// TIA Portal V16 export
// export: Created 2022-07-21T09:35:28.3226111Z, ExportSetting WithDefaults, DisplayName Totally Integrated Automation Portal, DisplayVersion V16 Update 4, DisplayName TIA Portal Version Control Interface, DisplayVersion V16 Update 2, DisplayName TIA Portal Openness, DisplayVersion V16 Update 4, DisplayName SINAMICS Startdrive Advanced, DisplayVersion V16 Update 5, DisplayName SINAMICS Startdrive G130, G150, S120, S150, SINAMICS MV, S210, DisplayVersion V16 Update 5, DisplayName SINAMICS Startdrive G110M, G120, G120C, G120D, G120P, G115D, DisplayVersion V16 Update 5, DisplayName STEP 7 Professional, DisplayVersion V16 Update 4, DisplayName STEP 7 Safety, DisplayVersion V16, DisplayName WinCC Advanced, DisplayVersion V16 Update 4
FUNCTION_BLOCK "fbDriveSiemens"   // FB706, LAD
TITLE = Drive Siemens
{ S7_Optimized_Access := 'TRUE' }
VERSION : 0.1
// stored: AutoNumber false, IsIECCheckEnabled false, IsRetainMemResEnabled false, MemoryReserve 100, SetENOAutomatically false, UDAEnableTagReadback false
   VAR_INPUT
      executeAbslute : Bool;   // Ruch do zadanej pozycji / Move to preset position
      executeRelative : Bool;   // Przesunięcie o zadaną pozycję / Move by preset position
      stop : Bool;   // stop
      extAlm : Bool;   // zewnętrzny alarm / external alarm
      velocityAuto : LReal;   // [mm/s]
      velocityMan : LReal;   // [mm/s]
      acceleration : LReal;   // [mm/s²]
      decceleration : LReal;   // [mm/s²]
      group : "typeGroup";
      axis : TO_PositioningAxis;
   END_VAR
   VAR_IN_OUT
      drive : "typeDrive";
      axisBasicsDataBlock : "LAxisBasics_typeAxisBasicsData";
      axisConfiguration : "LAxisCtrl_typeAxisConfig";
   END_VAR
   VAR
      delayPTAlm0 : Time := T#1s;   // Czas opóźnienia dla alarmu 0 / delay alarm 0
      delayPTAlm1 : Time := T#1s;   // Czas opóźnienia dla alarmu 1 / delay alarm 1
      delayPTAlm2 : Time := T#1s;   // Czas opóźnienia dla alarmu 2 / delay alarm 2
      delayPTAlm3 : Time := T#1s;   // Czas opóźnienia dla alarmu 3 / delay alarm 3
      delayPTAlm4 : Time := T#1s;   // Czas opóźnienia dla alarmu 4 / delay alarm 4
      delayPTAlm5 : Time := T#1s;   // Czas opóźnienia dla alarmu 5 / delay alarm 5
      delayPTAlm6 : Time := T#1s;   // Czas opóźnienia dla alarmu 6 / delay alarm 6
      delayPTAlm7 : Time := T#1s;   // Czas opóźnienia dla alarmu 7 / delay alarm 7
      instTmrDlyAlm0 { S7_SetPoint := 'True'} : TON_TIME;   // Opóźnienie dla alarmu 0 / delay alarm 0
      instTmrDlyAlm1 { S7_SetPoint := 'True'} : TON_TIME;   // Opóźnienie dla alarmu 1 / delay alarm 1
      instTmrDlyAlm2 { S7_SetPoint := 'True'} : TON_TIME;   // Opóźnienie dla alarmu 2 / delay alarm 2
      instTmrDlyAlm3 { S7_SetPoint := 'True'} : TON_TIME;   // Opóźnienie dla alarmu 3 / delay alarm 3
      instTmrDlyAlm4 { S7_SetPoint := 'True'} : TON_TIME;   // Opóźnienie dla alarmu 4 / delay alarm 4
      instTmrDlyAlm5 { S7_SetPoint := 'True'} : TON_TIME;   // Opóźnienie dla alarmu 5 / delay alarm 5
      instTmrDlyAlm6 { S7_SetPoint := 'True'} : TON_TIME;   // Opóźnienie dla alarmu 6 / delay alarm 6
      instTmrDlyAlm7 { S7_SetPoint := 'True'} : TON_TIME;   // Opóźnienie dla alarmu 7 / delay alarm 7
      instLAxisCtrl_PosAxis { S7_SetPoint := 'True'} : "LAxisCtrl_PosAxis";
      instSetpointVelocity { S7_SetPoint := 'True'} : "fbSPEntryLReal";
      instSetpointPosition { S7_SetPoint := 'True'} : "fbSPEntryLReal";
      statOldAuto { S7_SetPoint := 'True'} : Bool;
      statOldMan : Bool;
      homePulse { S7_SetPoint := 'True'} : TP_TIME;
      instCompPosHome { S7_SetPoint := 'True'} : "fbCompareLReal";   // Porównanie pozycji domowej oś Z / Compare home position Z axis
   END_VAR
   VAR_TEMP
      bAlm0 : Bool;   // tymczasowy bit dla alarmu 0 / temporary alarm bit 0
      bAlm1 : Bool;   // tymczasowy bit dla alarmu 1 / temporary alarm bit 1
      bAlm2 : Bool;   // tymczasowy bit dla alarmu 2 / temporary alarm bit 2
      bAlm3 : Bool;   // tymczasowy bit dla alarmu 3 / temporary alarm bit 3
      bAlm4 : Bool;   // tymczasowy bit dla alarmu 4 / temporary alarm bit 4
      bAlm5 : Bool;   // tymczasowy bit dla alarmu 5 / temporary alarm bit 5
      bAlm6 : Bool;   // tymczasowy bit dla alarmu 6 / temporary alarm bit 6
      bAlm7 : Bool;   // tymczasowy bit dla alarmu 7 / temporary alarm bit 7
      seqStart : Bool;
      "robot in cv zone" : Bool;
   END_VAR
   VAR CONSTANT
      MAX_VEL_AUTO : LReal := 2000.0;   // prędkość w trybie automatycznym / speed in automatic mode
      MAX_VEL_MAN : LReal := 2000.0;
      MIN_VEL : LReal := 0.1;
      MIN_DIST : LReal := -1000.0;
      MAX_DIST : LReal := 5000.0;
   END_VAR
BEGIN

REGION Network 1: Alarm: axis error / Alarm: błąd osi
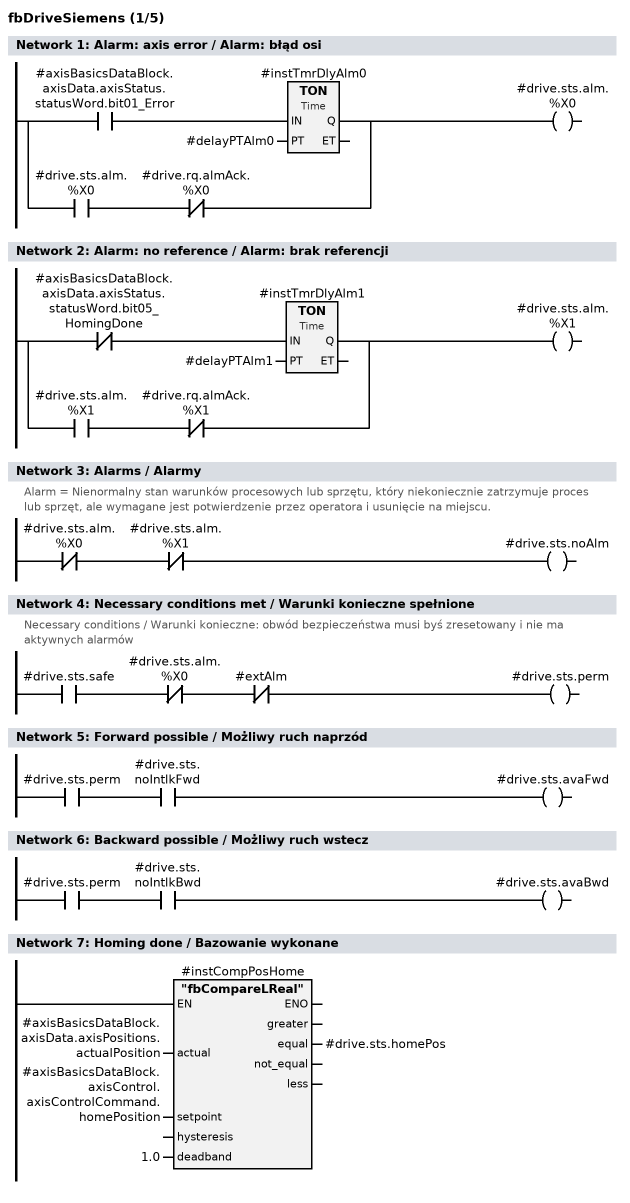
   RUNG wire#powerrail
      Contact( #axisBasicsDataBlock.axisData.axisStatus.statusWord.bit01_Error )
      { S7_Templates := "time_type := Time" } #instTmrDlyAlm0.TON(pt := #delayPTAlm0, et =>)
      wire#w1
      Coil( #drive.sts.alm.%X0 )
   END_RUNG
   RUNG wire#powerrail
      Contact( #drive.sts.alm.%X0 )
      I_Contact( #drive.rq.almAck.%X0 )
   END_RUNG wire#w1
   // the same network as SCL:
   #instTmrDlyAlm0(IN := #axisBasicsDataBlock.axisData.axisStatus.statusWord.bit01_Error, PT := #delayPTAlm0);   // TON
   #drive.sts.alm.%X0 := #instTmrDlyAlm0.Q OR (#drive.sts.alm.%X0 AND NOT #drive.rq.almAck.%X0);
END_REGION

REGION Network 2: Alarm: no reference / Alarm: brak referencji
   RUNG wire#powerrail
      I_Contact( #axisBasicsDataBlock.axisData.axisStatus.statusWord.bit05_HomingDone )
      { S7_Templates := "time_type := Time" } #instTmrDlyAlm1.TON(pt := #delayPTAlm1, et =>)
      wire#w1
      Coil( #drive.sts.alm.%X1 )
   END_RUNG
   RUNG wire#powerrail
      Contact( #drive.sts.alm.%X1 )
      I_Contact( #drive.rq.almAck.%X1 )
   END_RUNG wire#w1
   // the same network as SCL:
   #instTmrDlyAlm1(IN := NOT #axisBasicsDataBlock.axisData.axisStatus.statusWord.bit05_HomingDone,   // TON
                   PT := #delayPTAlm1);
   #drive.sts.alm.%X1 := #instTmrDlyAlm1.Q OR (#drive.sts.alm.%X1 AND NOT #drive.rq.almAck.%X1);
END_REGION

REGION Network 3: Alarms / Alarmy
   // Alarm = Nienormalny stan warunków procesowych lub sprzętu, który niekoniecznie zatrzymuje proces lub sprzęt, ale wymagane jest potwierdzenie przez operatora i usunięcie na miejscu.
   RUNG wire#powerrail
      I_Contact( #drive.sts.alm.%X0 )
      I_Contact( #drive.sts.alm.%X1 )
      Coil( #drive.sts.noAlm )
   END_RUNG
   // the same network as SCL:
   #drive.sts.noAlm := NOT #drive.sts.alm.%X0 AND NOT #drive.sts.alm.%X1;
END_REGION

REGION Network 4: Necessary conditions met / Warunki konieczne spełnione
   // Necessary conditions / Warunki konieczne: obwód bezpieczeństwa musi byś zresetowany i nie ma aktywnych alarmów
   RUNG wire#powerrail
      Contact( #drive.sts.safe )
      I_Contact( #drive.sts.alm.%X0 )
      I_Contact( #extAlm )
      Coil( #drive.sts.perm )
   END_RUNG
   // the same network as SCL:
   #drive.sts.perm := #drive.sts.safe AND NOT #drive.sts.alm.%X0 AND NOT #extAlm;
END_REGION

REGION Network 5: Forward possible / Możliwy ruch naprzód
   RUNG wire#powerrail
      Contact( #drive.sts.perm )
      Contact( #drive.sts.noIntlkFwd )
      Coil( #drive.sts.avaFwd )
   END_RUNG
   // the same network as SCL:
   #drive.sts.avaFwd := #drive.sts.perm AND #drive.sts.noIntlkFwd;
END_REGION

REGION Network 6: Backward possible / Możliwy ruch wstecz
   RUNG wire#powerrail
      Contact( #drive.sts.perm )
      Contact( #drive.sts.noIntlkBwd )
      Coil( #drive.sts.avaBwd )
   END_RUNG
   // the same network as SCL:
   #drive.sts.avaBwd := #drive.sts.perm AND #drive.sts.noIntlkBwd;
END_REGION

REGION Network 7: Homing done / Bazowanie wykonane
   RUNG wire#powerrail
      #instCompPosHome(actual := #axisBasicsDataBlock.axisData.axisPositions.actualPosition, setpoint := #axisBasicsDataBlock.axisControl.axisControlCommand.homePosition, hysteresis :=, deadband := 1.0, greater =>, equal => #drive.sts.homePos, not_equal =>, less =>)
   END_RUNG
   // the same network as SCL:
   #instCompPosHome(actual := #axisBasicsDataBlock.axisData.axisPositions.actualPosition,   // "fbCompareLReal"
                    setpoint := #axisBasicsDataBlock.axisControl.axisControlCommand.homePosition,
                    deadband := 1.0,
                    equal => #drive.sts.homePos);
END_REGION

REGION Network 8: Enable / Zezwolenie
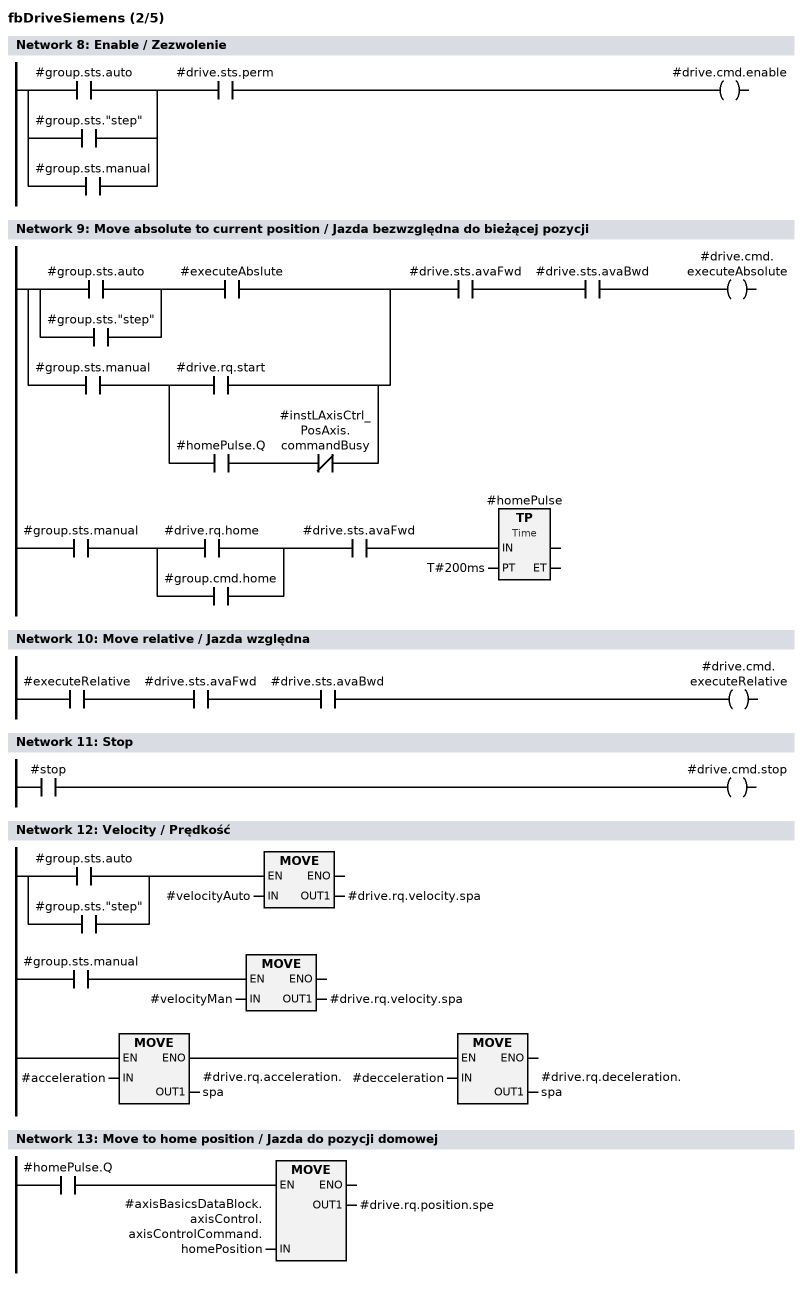
   RUNG wire#powerrail
      Contact( #group.sts.auto )
      wire#w1
      Contact( #drive.sts.perm )
      Coil( #drive.cmd.enable )
   END_RUNG
   RUNG wire#powerrail
      Contact( #group.sts."step" )
   END_RUNG wire#w1
   RUNG wire#powerrail
      Contact( #group.sts.manual )
   END_RUNG wire#w1
   // the same network as SCL:
   #drive.cmd.enable := (#group.sts.auto OR #group.sts."step" OR #group.sts.manual) AND #drive.sts.perm;
END_REGION

REGION Network 9: Move absolute to current position / Jazda bezwzględna do bieżącej pozycji
   RUNG wire#powerrail
      Contact( #group.sts.auto )
      wire#w1
      Contact( #executeAbslute )
      wire#w2
      Contact( #drive.sts.avaFwd )
      Contact( #drive.sts.avaBwd )
      Coil( #drive.cmd.executeAbsolute )
   END_RUNG
   RUNG wire#powerrail
      Contact( #group.sts."step" )
   END_RUNG wire#w1
   RUNG wire#powerrail
      Contact( #group.sts.manual )
      wire#w3
      Contact( #drive.rq.start )
   END_RUNG wire#w2
   RUNG wire#w3
      Contact( #homePulse.Q )
      I_Contact( #instLAxisCtrl_PosAxis.commandBusy )
   END_RUNG wire#w2
   RUNG wire#powerrail
      Contact( #group.sts.manual )
      wire#w4
      Contact( #drive.rq.home )
      wire#w5
      Contact( #drive.sts.avaFwd )
      { S7_Templates := "time_type := Time" } #homePulse.TP(pt := T#200ms, et =>)
   END_RUNG
   RUNG wire#w4
      Contact( #group.cmd.home )
   END_RUNG wire#w5
   // the same network as SCL:
   #drive.cmd.executeAbsolute := (((#group.sts.auto OR #group.sts."step") AND #executeAbslute) OR (#group.sts.manual AND (#drive.rq.start OR (#homePulse.Q AND NOT #instLAxisCtrl_PosAxis.commandBusy)))) AND #drive.sts.avaFwd AND #drive.sts.avaBwd;
   #homePulse(IN := #group.sts.manual AND (#drive.rq.home OR #group.cmd.home) AND #drive.sts.avaFwd,   // TP
              PT := T#200ms);
END_REGION

REGION Network 10: Move relative / Jazda względna
   RUNG wire#powerrail
      Contact( #executeRelative )
      Contact( #drive.sts.avaFwd )
      Contact( #drive.sts.avaBwd )
      Coil( #drive.cmd.executeRelative )
   END_RUNG
   // the same network as SCL:
   #drive.cmd.executeRelative := #executeRelative AND #drive.sts.avaFwd AND #drive.sts.avaBwd;
END_REGION

REGION Network 11: Stop
   RUNG wire#powerrail
      Contact( #stop )
      Coil( #drive.cmd.stop )
   END_RUNG
   // the same network as SCL:
   #drive.cmd.stop := #stop;
END_REGION

REGION Network 12: Velocity / Prędkość
   RUNG wire#powerrail
      Contact( #group.sts.auto )
      wire#w1
      Move(in := #velocityAuto, out1 => #drive.rq.velocity.spa)
   END_RUNG
   RUNG wire#powerrail
      Contact( #group.sts."step" )
   END_RUNG wire#w1
   RUNG wire#powerrail
      Contact( #group.sts.manual )
      Move(in := #velocityMan, out1 => #drive.rq.velocity.spa)
   END_RUNG
   RUNG wire#powerrail
      Move(in := #acceleration, out1 => #drive.rq.acceleration.spa)
      Move(in := #decceleration, out1 => #drive.rq.deceleration.spa)
   END_RUNG
   // the same network as SCL:
   IF #group.sts.auto OR #group.sts."step" THEN #drive.rq.velocity.spa := #velocityAuto; END_IF;
   IF #group.sts.manual THEN #drive.rq.velocity.spa := #velocityMan; END_IF;
   #drive.rq.acceleration.spa := #acceleration;
   #drive.rq.deceleration.spa := #decceleration;
END_REGION

REGION Network 13: Move to home position / Jazda do pozycji domowej
   RUNG wire#powerrail
      Contact( #homePulse.Q )
      Move(in := #axisBasicsDataBlock.axisControl.axisControlCommand.homePosition, out1 => #drive.rq.position.spe)
   END_RUNG
   // the same network as SCL:
   IF #homePulse.Q THEN
       #drive.rq.position.spe := #axisBasicsDataBlock.axisControl.axisControlCommand.homePosition;
   END_IF;
END_REGION

REGION Network 14: Velocity change depending on selected mode / Zmiana prędkości w zależności od trybu sterowania
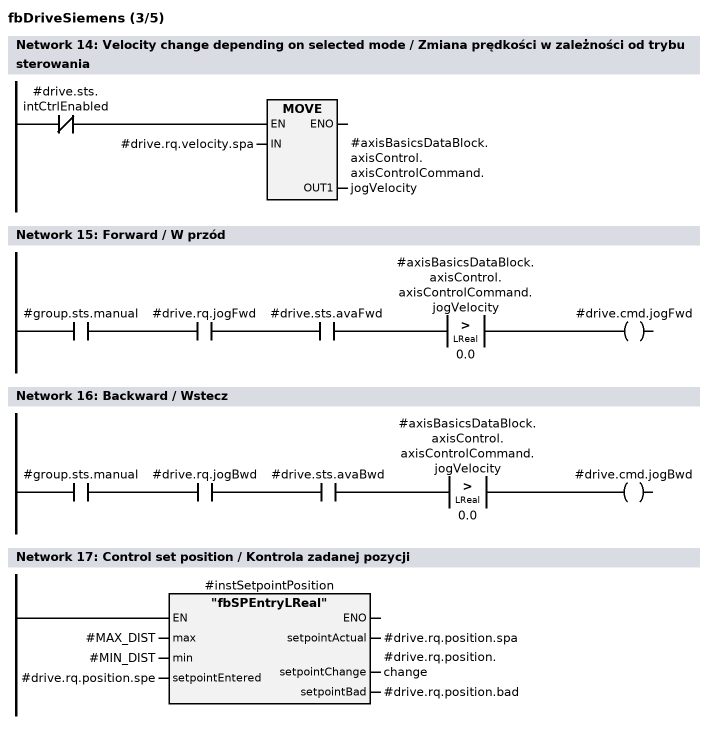
   RUNG wire#powerrail
      I_Contact( #drive.sts.intCtrlEnabled )
      Move(in := #drive.rq.velocity.spa, out1 => #axisBasicsDataBlock.axisControl.axisControlCommand.jogVelocity)
   END_RUNG
   // the same network as SCL:
   IF NOT #drive.sts.intCtrlEnabled THEN
       #axisBasicsDataBlock.axisControl.axisControlCommand.jogVelocity := #drive.rq.velocity.spa;
   END_IF;
END_REGION

REGION Network 15: Forward / W przód
   RUNG wire#powerrail
      Contact( #group.sts.manual )
      Contact( #drive.rq.jogFwd )
      Contact( #drive.sts.avaFwd )
      { S7_Templates := "SrcType := LReal" } GT_Contact(in1 := #axisBasicsDataBlock.axisControl.axisControlCommand.jogVelocity, in2 := 0.0)
      Coil( #drive.cmd.jogFwd )
   END_RUNG
   // the same network as SCL:
   #drive.cmd.jogFwd := #group.sts.manual AND #drive.rq.jogFwd AND #drive.sts.avaFwd AND (#axisBasicsDataBlock.axisControl.axisControlCommand.jogVelocity > 0.0);
END_REGION

REGION Network 16: Backward / Wstecz
   RUNG wire#powerrail
      Contact( #group.sts.manual )
      Contact( #drive.rq.jogBwd )
      Contact( #drive.sts.avaBwd )
      { S7_Templates := "SrcType := LReal" } GT_Contact(in1 := #axisBasicsDataBlock.axisControl.axisControlCommand.jogVelocity, in2 := 0.0)
      Coil( #drive.cmd.jogBwd )
   END_RUNG
   // the same network as SCL:
   #drive.cmd.jogBwd := #group.sts.manual AND #drive.rq.jogBwd AND #drive.sts.avaBwd AND (#axisBasicsDataBlock.axisControl.axisControlCommand.jogVelocity > 0.0);
END_REGION

REGION Network 17: Control set position / Kontrola zadanej pozycji
   RUNG wire#powerrail
      #instSetpointPosition(max := #MAX_DIST, min := #MIN_DIST, setpointEntered := #drive.rq.position.spe, setpointActual => #drive.rq.position.spa, setpointChange => #drive.rq.position.change, setpointBad => #drive.rq.position.bad)
   END_RUNG
   // the same network as SCL:
   #instSetpointPosition(max := #MAX_DIST,   // "fbSPEntryLReal"
                         min := #MIN_DIST,
                         setpointEntered := #drive.rq.position.spe,
                         setpointActual => #drive.rq.position.spa,
                         setpointChange => #drive.rq.position.change,
                         setpointBad => #drive.rq.position.bad);
END_REGION

REGION Network 18 (SCL): Parameters for control block / Parametry dla bloczka sterowania
   //power
   #axisConfiguration.power.startMode := #axisBasicsDataBlock.axisControl.axisControlCommand.powerStartMode; //1
   #axisConfiguration.power.stopMode := #axisBasicsDataBlock.axisControl.axisControlCommand.powerStopMode;

   //reset
   #axisConfiguration.generalSettings.resetWithRestart := #axisBasicsDataBlock.axisControl.axisControlCommand.resetRestart;

   //jog mode
   #axisConfiguration.jog.velocity := #axisBasicsDataBlock.axisControl.axisControlCommand.jogVelocity;
   #axisConfiguration.jog.acceleration := #axisBasicsDataBlock.axisControl.axisControlCommand.jogAcceleration;
   #axisConfiguration.jog.deceleration := #axisBasicsDataBlock.axisControl.axisControlCommand.jogDeceleration;
   #axisConfiguration.jog.jerk := #axisBasicsDataBlock.axisControl.axisControlCommand.jogJerk;
   #axisConfiguration.jog.increment := 1;
   #axisConfiguration.jog.positionControlled := #axisBasicsDataBlock.axisControl.axisControlCommand.jogPositionControlled;

   //homing 
   #axisConfiguration.homing.mode := #axisBasicsDataBlock.axisControl.axisControlCommand.homeMode; //7; 
   #axisConfiguration.homing.position := #axisBasicsDataBlock.axisControl.axisControlCommand.homePosition; //0;
   #axisConfiguration.homing.extendedMode := -1; //no extended mode

   //posAbsolute
   #axisConfiguration.posAbsolute.velocity := #drive.rq.velocity.spa;
   #axisConfiguration.posAbsolute.position := #drive.rq.position.spa;
   #axisConfiguration.posAbsolute.acceleration := #drive.rq.acceleration.spa;
   #axisConfiguration.posAbsolute.deceleration := #drive.rq.deceleration.spa;
   #axisConfiguration.posAbsolute.jerk := #axisConfiguration.jog.jerk;
   #axisConfiguration.posAbsolute.direction := 1; 

   //posRelative
   #axisConfiguration.posRelative.velocity := #drive.rq.velocity.spa;
   #axisConfiguration.posRelative.acceleration := #drive.rq.acceleration.spa;
   #axisConfiguration.posRelative.deceleration := #drive.rq.deceleration.spa;
   #axisConfiguration.posRelative.jerk := #axisConfiguration.jog.jerk;
   #axisConfiguration.posRelative.distance := #drive.rq.position.spa;
   #axisConfiguration.posRelative.direction := 0; //---> kierunek wyznaczony na podstawie "distance"
END_REGION

REGION Network 19: Control block / Bloczek sterowania
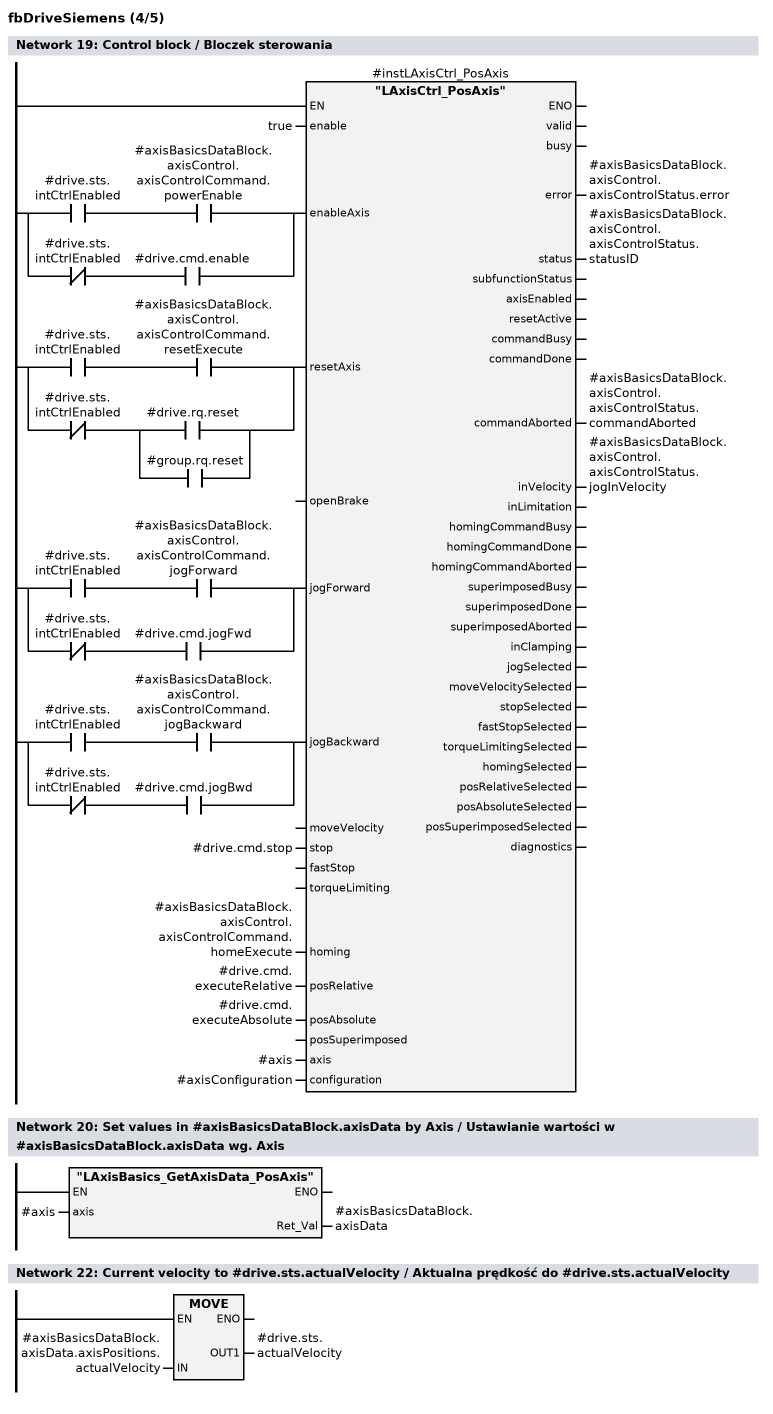
   RUNG wire#powerrail
      #instLAxisCtrl_PosAxis(enableAxis := wire#w1, resetAxis := wire#w3, jogForward := wire#w4, jogBackward := wire#w5, enable := true, openBrake :=, moveVelocity :=, stop := #drive.cmd.stop, fastStop :=, torqueLimiting :=, homing := #axisBasicsDataBlock.axisControl.axisControlCommand.homeExecute, posRelative := #drive.cmd.executeRelative, posAbsolute := #drive.cmd.executeAbsolute, posSuperimposed :=, axis := #axis, configuration := #axisConfiguration, valid =>, busy =>, error => #axisBasicsDataBlock.axisControl.axisControlStatus.error, status => #axisBasicsDataBlock.axisControl.axisControlStatus.statusID, subfunctionStatus =>, axisEnabled =>, resetActive =>, commandBusy =>, commandDone =>, commandAborted => #axisBasicsDataBlock.axisControl.axisControlStatus.commandAborted, inVelocity => #axisBasicsDataBlock.axisControl.axisControlStatus.jogInVelocity, inLimitation =>, homingCommandBusy =>, homingCommandDone =>, homingCommandAborted =>, superimposedBusy =>, superimposedDone =>, superimposedAborted =>, inClamping =>, jogSelected =>, moveVelocitySelected =>, stopSelected =>, fastStopSelected =>, torqueLimitingSelected =>, homingSelected =>, posRelativeSelected =>, posAbsoluteSelected =>, posSuperimposedSelected =>, diagnostics =>)
   END_RUNG
   RUNG wire#powerrail
      Contact( #drive.sts.intCtrlEnabled )
      Contact( #axisBasicsDataBlock.axisControl.axisControlCommand.powerEnable )
   END_RUNG wire#w1
   RUNG wire#powerrail
      I_Contact( #drive.sts.intCtrlEnabled )
      Contact( #drive.cmd.enable )
   END_RUNG wire#w1
   RUNG wire#powerrail
      Contact( #drive.sts.intCtrlEnabled )
      Contact( #axisBasicsDataBlock.axisControl.axisControlCommand.resetExecute )
   END_RUNG wire#w3
   RUNG wire#powerrail
      I_Contact( #drive.sts.intCtrlEnabled )
      wire#w2
      Contact( #drive.rq.reset )
   END_RUNG wire#w3
   RUNG wire#w2
      Contact( #group.rq.reset )
   END_RUNG wire#w3
   RUNG wire#powerrail
      Contact( #drive.sts.intCtrlEnabled )
      Contact( #axisBasicsDataBlock.axisControl.axisControlCommand.jogForward )
   END_RUNG wire#w4
   RUNG wire#powerrail
      I_Contact( #drive.sts.intCtrlEnabled )
      Contact( #drive.cmd.jogFwd )
   END_RUNG wire#w4
   RUNG wire#powerrail
      Contact( #drive.sts.intCtrlEnabled )
      Contact( #axisBasicsDataBlock.axisControl.axisControlCommand.jogBackward )
   END_RUNG wire#w5
   RUNG wire#powerrail
      I_Contact( #drive.sts.intCtrlEnabled )
      Contact( #drive.cmd.jogBwd )
   END_RUNG wire#w5
   // the same network as SCL:
   #instLAxisCtrl_PosAxis(enable := true,   // "LAxisCtrl_PosAxis"
                          enableAxis := (#drive.sts.intCtrlEnabled AND #axisBasicsDataBlock.axisControl.axisControlCommand.powerEnable) OR (NOT #drive.sts.intCtrlEnabled AND #drive.cmd.enable),
                          resetAxis := (#drive.sts.intCtrlEnabled AND #axisBasicsDataBlock.axisControl.axisControlCommand.resetExecute) OR (NOT #drive.sts.intCtrlEnabled AND (#drive.rq.reset OR #group.rq.reset)),
                          jogForward := (#drive.sts.intCtrlEnabled AND #axisBasicsDataBlock.axisControl.axisControlCommand.jogForward) OR (NOT #drive.sts.intCtrlEnabled AND #drive.cmd.jogFwd),
                          jogBackward := (#drive.sts.intCtrlEnabled AND #axisBasicsDataBlock.axisControl.axisControlCommand.jogBackward) OR (NOT #drive.sts.intCtrlEnabled AND #drive.cmd.jogBwd),
                          stop := #drive.cmd.stop,
                          homing := #axisBasicsDataBlock.axisControl.axisControlCommand.homeExecute,
                          posRelative := #drive.cmd.executeRelative,
                          posAbsolute := #drive.cmd.executeAbsolute,
                          axis := #axis,
                          configuration := #axisConfiguration,
                          error => #axisBasicsDataBlock.axisControl.axisControlStatus.error,
                          status => #axisBasicsDataBlock.axisControl.axisControlStatus.statusID,
                          commandAborted => #axisBasicsDataBlock.axisControl.axisControlStatus.commandAborted,
                          inVelocity => #axisBasicsDataBlock.axisControl.axisControlStatus.jogInVelocity);
END_REGION

REGION Network 20: Set values in #axisBasicsDataBlock.axisData by Axis / Ustawianie wartości w #axisBasicsDataBlock.axisData wg. Axis
   RUNG wire#powerrail
      "LAxisBasics_GetAxisData_PosAxis"(axis := #axis, Ret_Val => #axisBasicsDataBlock.axisData)
   END_RUNG
   // the same network as SCL:
   #axisBasicsDataBlock.axisData := "LAxisBasics_GetAxisData_PosAxis"(axis := #axis);
END_REGION

REGION Network 21 (SCL): Set values in #axisBasicsDataBlock.axisData / Ustawianie wartości w #axisBasicsDataBlock.axisData

   #axisBasicsDataBlock.axisControl.axisControlStatus.powerStatus := #instLAxisCtrl_PosAxis.instPower.Status;
   #axisBasicsDataBlock.axisControl.axisControlStatus.powerBusy := #instLAxisCtrl_PosAxis.instPower.Busy;
   #axisBasicsDataBlock.axisControl.axisControlStatus.resetDone := #instLAxisCtrl_PosAxis.instReset.Done;
   #axisBasicsDataBlock.axisControl.axisControlStatus.resetBusy := #instLAxisCtrl_PosAxis.instReset.Busy;

   #axisBasicsDataBlock.axisControl.axisControlStatus.jogBusy := #instLAxisCtrl_PosAxis.instMoveJog.Busy;
   #axisBasicsDataBlock.axisControl.axisControlStatus.homeBusy := #instLAxisCtrl_PosAxis.instHome.Busy;
   #axisBasicsDataBlock.axisControl.axisControlStatus.homeDone := #instLAxisCtrl_PosAxis.instHome.Done;

   #axisBasicsDataBlock.moveToEndPos.moveToEndPosStatus.inPosition := #instLAxisCtrl_PosAxis.instMoveAbsolute.Done;

   #instLAxisCtrl_PosAxis.instHome.Error := #instLAxisCtrl_PosAxis.instHome.Error;
   #instLAxisCtrl_PosAxis.instHome.ErrorId := #instLAxisCtrl_PosAxis.instHome.ErrorId;
END_REGION

REGION Network 22: Current velocity to #drive.sts.actualVelocity / Aktualna prędkość do #drive.sts.actualVelocity
   RUNG wire#powerrail
      Move(in := #axisBasicsDataBlock.axisData.axisPositions.actualVelocity, out1 => #drive.sts.actualVelocity)
   END_RUNG
   // the same network as SCL:
   #drive.sts.actualVelocity := #axisBasicsDataBlock.axisData.axisPositions.actualVelocity;
END_REGION

REGION Network 23: Current position to #drive.sts.actualPosition / Aktualna pozycja do #drive.sts.actualPosition
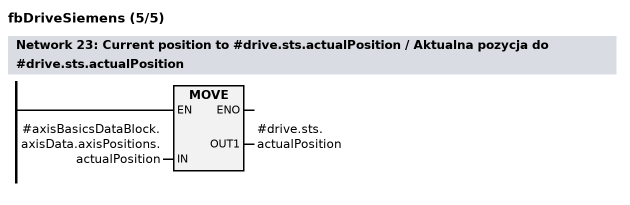
   RUNG wire#powerrail
      Move(in := #axisBasicsDataBlock.axisData.axisPositions.actualPosition, out1 => #drive.sts.actualPosition)
   END_RUNG
   // the same network as SCL:
   #drive.sts.actualPosition := #axisBasicsDataBlock.axisData.axisPositions.actualPosition;
END_REGION
END_FUNCTION_BLOCK
